FUNCTION f_To_T_Process : T_process
VAR_INPUT
  nExp              : BYTE;
END_VAR
VAR
  rVal              : LREAL;
  nTmp              : ULINT; 
  wTmp              : T_PROCESS;
END_VAR

rVal   := TO_LREAL(SEL(nExp > SIZEOF(T_PROCESS)*8, nExp, SIZEOF(T_PROCESS)*8));
nTmp   := TO_ULINT(EXPT(2,rVal)-1);

memcpy(ADR(wtmp), ADR(ntmp), SIZEOF(wtmp));

f_To_T_Process      := wtmp;

END_FUNCTION

(* stored: Version 1.1.0.1
   POU f_To_T_Process: Id {60bbd1c1-ea14-4596-88bd-c1007ec08aa7}, SpecialFunc None *)
